SUBAPPLICATION Uebung_001d2_AX (* DigitalInput_I1/2 auf DigitalOutput_Q1/2, als Alternative(Verriegelt) mit Plug and Socket, ohne ECC *)
  (* Standard: 61499-2; Description: Copyright (c) 2023 Meisterschulen am Ostbahnhof This program and the accompanying materials are made available under the terms of the Eclipse Public License 2.0 which is available at https://www.eclipse.org/legal/epl-2.0/ SPDX-License-Identifier: EPL-2.0 *)
  (* Version 1.0, 2023-10-23, Franz Höpfinger, Meisterschulen am Ostbahnhof, initial API and implementation and/or initial documentation *)
  PACKAGE Uebungen;
  IMPORT logiBUS::io::DI::logiBUS_DI::Input_I1;
  IMPORT logiBUS::io::DI::logiBUS_DI::Input_I2;
  IMPORT logiBUS::io::DQ::logiBUS_DO::Output_Q1;
  IMPORT logiBUS::io::DQ::logiBUS_DO::Output_Q2;
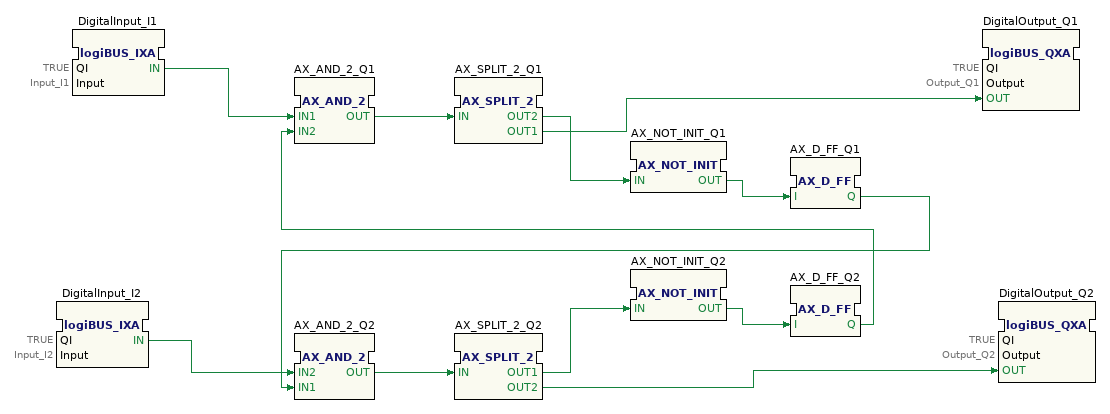
  (* Kompliziert. BESSER: ILOCK-Baustein *)
  FBS
    DigitalInput_I1 : logiBUS::io::DI::logiBUS_IXA(QI := TRUE, Input := Input_I1);
    DigitalOutput_Q1 : logiBUS::io::DQ::logiBUS_QXA(QI := TRUE, Output := Output_Q1);
    AX_AND_2_Q1 : adapter::booleanOperators::AX_AND_2;
    DigitalOutput_Q2 : logiBUS::io::DQ::logiBUS_QXA(QI := TRUE, Output := Output_Q2);
    AX_AND_2_Q2 : adapter::booleanOperators::AX_AND_2;
    DigitalInput_I2 : logiBUS::io::DI::logiBUS_IXA(QI := TRUE, Input := Input_I2);
    AX_SPLIT_2_Q1 : adapter::events::unidirectional::AX_SPLIT_2;
    AX_SPLIT_2_Q2 : adapter::events::unidirectional::AX_SPLIT_2;
    AX_NOT_INIT_Q1 : adapter::booleanOperators::AX_NOT_INIT;
    AX_NOT_INIT_Q2 : adapter::booleanOperators::AX_NOT_INIT;
    AX_D_FF_Q1 : adapter::events::unidirectional::AX_D_FF;
    AX_D_FF_Q2 : adapter::events::unidirectional::AX_D_FF;
  END_FBS
  ADAPTER_CONNECTIONS
    AX_AND_2_Q1.OUT TO AX_SPLIT_2_Q1.IN;
    AX_AND_2_Q2.OUT TO AX_SPLIT_2_Q2.IN;
    AX_SPLIT_2_Q1.OUT2 TO AX_NOT_INIT_Q1.IN;
    AX_SPLIT_2_Q2.OUT1 TO AX_NOT_INIT_Q2.IN;
    DigitalInput_I2.IN TO AX_AND_2_Q2.IN2;
    AX_SPLIT_2_Q2.OUT2 TO DigitalOutput_Q2.OUT;
    AX_SPLIT_2_Q1.OUT1 TO DigitalOutput_Q1.OUT;
    DigitalInput_I1.IN TO AX_AND_2_Q1.IN1;
    AX_NOT_INIT_Q2.OUT TO AX_D_FF_Q2.I;
    AX_NOT_INIT_Q1.OUT TO AX_D_FF_Q1.I;
    AX_D_FF_Q1.Q TO AX_AND_2_Q2.IN1;
    AX_D_FF_Q2.Q TO AX_AND_2_Q1.IN2;
  END_CONNECTIONS
END_SUBAPPLICATION
